// TwinCAT 3 PLC project POS_Temp_system
// ProgramVersion: 3.1.4022.3
// libraries:
//   CAA Types Extern, * (CAA Technical Workgroup)
//   Tc2_ControllerToolbox, * (Beckhoff Automation GmbH)
//   Tc2_Standard, * (Beckhoff Automation GmbH)
//   Tc2_System, * (Beckhoff Automation GmbH)
//   Tc2_Utilities, * (Beckhoff Automation GmbH)
//   Tc3_Module, * (Beckhoff Automation GmbH)
//   VisuSymbols,3.5.10.0,System
// project tree:
//   DUTs/ SeqState.TcTLEO (not stored)
//   fbBLOCKS/ fBDISCRETE_PID.TcPOU, fbSensorNoise.TcPOU, FirstOrder.TcPOU
//   / GlobalTextList.TcGTLO, PlcTask.TcTTO (not stored), Visualization Manager.TcVMO (not stored)
//   GVLs/ GVL_IO.TcGVL
//   POUs/ MAIN.TcPOU
//   PROCESSES/ HEATER_PROCESS.TcPOU, SERVO_POS.TcPOU, TANKLEVEL.TcPOU
//   VISUs/ UserInterface.TcVIS

// ---- GVLs/GVL_IO.TcGVL
{attribute 'qualified_only'}
VAR_GLOBAL
// Process parameters, variables	
	SetPoint_ServoX           :REAL;      // SetPoint X - axis
	SetPointHeater            :REAL;      // SetPoint Heater
	Output_ServoX             :REAL;      // X-axis Position
	Output_Heater             :REAL;      // Temperature Heater
	Output_Stirrer            :BOOL;      // Mixer / Stirrer 
	TankLevelSensor           :REAL;      // Tanklevel analogue sensor 
	ValveA, ValveB, ValveC    :BOOL;      // Valves
	Stirrer					  :BOOL;	  // activate stirrer
	xPushButton1              :BOOL;      // Used for test purposes 
	xPushButton2              :BOOL;      // Used for test purposes
	StartPr, StopPr           :BOOL;      // Start and Stop Process Buttons
	Level_S1,Level_S2,Level_S3:BOOL;      // Level Sensors (digital sensors)
    xGenCtrl_Error            :BOOL;      // General Error due SERVO or HEATER Control  
	//  
    noise_HeaterSensor        :BOOL;      // Sensor noise simulation on  
	noise_ServoSensor         :BOOL;      // Sensor noise simulation on          
	END_VAR

// ---- PROCESSES/TANKLEVEL.TcPOU
PROGRAM TANKLEVEL
VAR CONSTANT
	L_S1:REAL :=  5.00 ;
	L_S2:REAL := 60.00 ;
	L_S3:REAL := 80.00 ;	
END_VAR

VAR
	Plant:FirstOrder;
	//fbNoise : FB_CTRL_NOISE_GENERATOR ;
	//fbNoiseParams : ST_CTRL_NOISE_GENERATOR_PARAMS ;
	//noise_level : LREAL ;
	fill_ValveA,fill_ValveB,Drain_ValveC: BOOL;
	fbdelayOFF:TOF;
// ---	
    fbFill, fbDrain : R_TRIG;
	fbFillOff, fbDrainOff :F_TRIG;
	currConstTime: REAL := 15;
	spLevel : REAL:=0;
    SensorNoise:fbSensorNoise;
END_VAR

// Generate sensor noise
//fbNoiseParams . tCtrlCycleTime := T#10MS ;
//fbNoiseParams . tTaskCycleTime := T#10MS ;
//fbNoiseParams . fAmplitude := 1.5 ;
//fbNoise ( fManSyncValue := 1 , eMode := 2 , stParams := fbNoiseParams ) ;
//noise_level := fbNoise.fOut ;
// Valves
Fill_ValveA := GVL_IO.ValveA ;
Fill_ValveB := GVL_IO.ValveB ;
Drain_ValveC := GVL_IO.ValveC ;

fbFill(clk := ( Fill_ValveA XOR Fill_ValveB ) AND NOT Drain_ValveC ) ;
fbFillOff(clk := Fill_ValveA XOR Fill_ValveB ) ;
fbDrain(clk := Drain_ValveC );
fbDrainOff(clk := Drain_ValveC );
fbdelayOFF(IN:=(GVL_IO.ValveA OR GVL_IO.ValveB OR GVL_IO.ValveC),PT:=T#1S);

IF fbFill.Q THEN
	spLevel:=150;
	currConstTime:=15;
END_IF
IF fbFillOff.Q THEN
	spLevel:=plant.fBOut;
	
END_IF
IF fbDrain.Q THEN
	currConstTime:=5;
    spLevel:=1;	
END_IF

IF fbDrainOff.Q THEN
	spLevel := GVL_IO.TankLevelSensor ;
END_IF

Plant(fBIn:= spLevel,Gain := 1,Tconstant := currConstTime);
SensorNoise(noise_enable:=TRUE,Ampl:=1.0);
//GVL_IO.TankLevelSensor:=plant.fBOut;
GVL_IO.TankLevelSensor:=LREAL_TO_REAL(plant.fBOut +SensorNoise.noise_level);
// IF (fbdelayOFF.Q) THEN
//	GVL_IO.TankLevelSensor:=LREAL_TO_REAL(plant.fBOut +SensorNoise.noise_level);
// END_IF
GVL_IO.Level_S1:=TRUE;
GVL_IO.Level_S2:=TRUE;
GVL_IO.Level_S3:=TRUE;

IF GVL_IO.TankLevelSensor > L_S1 THEN
	GVL_IO.Level_S1:=FALSE;
END_IF
IF GVL_IO.TankLevelSensor > L_S2 THEN
	GVL_IO.Level_S2:=FALSE;
END_IF
IF GVL_IO.TankLevelSensor > L_S3 THEN
	GVL_IO.Level_S3:=FALSE;
END_IF

 //

END_PROGRAM

// ---- fbBLOCKS/FirstOrder.TcPOU
FUNCTION_BLOCK FirstOrder
VAR_INPUT
	Gain: REAL;
	Tconstant : REAL;
	fBIn   : REAL;
END_VAR
VAR_OUTPUT
	fBOut  : REAL;
END_VAR
VAR
	ssy, Sy   :REAL;
	Tsample: REAL := 0.01;
END_VAR

// This program simulates a First Order Euler Emulation
// Another way to simulate processes
// PLEASE DON'T CHANGE THE CODE IN THIS PROGRAM !
// Euler Emulation 1st Order with 0.01 sec sampletime.
sy := ( fBIn * Gain / Tconstant ) - ( fBOut / Tconstant ) ;
fBOut := fBout + ( sy * Tsample ) ;

END_FUNCTION_BLOCK

// ---- fbBLOCKS/fbSensorNoise.TcPOU
FUNCTION_BLOCK fbSensorNoise
VAR_INPUT
	noise_enable:BOOL;
	Ampl        :LREAL;
END_VAR
VAR_OUTPUT
noise_level : LREAL:=0;	
END_VAR
VAR
	fBNoise:FB_CTRL_NOISE_GENERATOR;
	fbNoiseParams: ST_CTRL_NOISE_GENERATOR_PARAMS;
END_VAR

// Generate noise for Sensors ( simulation ) 
fbNoiseParams.tCtrlCycleTime := T#10MS ;
fbNoiseParams.tTaskCycleTime := T#10MS ;
fbNoiseParams.fAmplitude := Ampl;

//
noise_level:=0;
IF Noise_enable THEN
	fbNoise ( fManSyncValue := 1 , eMode := 2 , stParams := fbNoiseParams ) ;
END_IF
noise_level:=fbNoise.fOut;

END_FUNCTION_BLOCK

// ---- fbBLOCKS/fBDISCRETE_PID.TcPOU
FUNCTION_BLOCK fBDISCRETE_PID
VAR_INPUT
	Setpoint       :REAL;   // SetPoint
    Kp             : REAL;  // Kp  Proportional gain
	Ki             : REAL;  // Ki  Integrated gain
	Kd             : REAL;  // Kd  Derivative gain
	Nfilter        : REAL;  // Lowpass Filter Coeff 
	Yprocess_value : REAL;  // Process Output
	Auto_Mode      : BOOL;  // PId enable if true (closed loop )
	MV_max_sat     : REAL;  // Maximum Saturation
	MV_min_sat     : REAL;  // Minimum Saturation
	//xExt_Error     : BOOL;  // External error 
	
END_VAR
VAR_OUTPUT
	MV_out        : REAL;    // Controller output
	Inposition    : BOOL;    //  2% Settled. is not implemented yet. 
END_VAR
VAR
	T1     : REAL :=0;
	Perr, Perr1, Perr2 : REAL ;
	deltaSetpoint :REAL;
    A,B,C  :REAL;
	MV_out1:REAL;
	Tsample:REAL := 0.01;
END_VAR

//
IF T1 = 0 THEN
	MV_out:=0;     // no bias offset  
END_IF
T1:=Tsample; 
Perr:= Setpoint - Yprocess_value; // Current error e[k]
// Check also PowerPoint Presentation module 5 
// Constant Coefficients including the Parameters Kp , Ki, Kd and Tsample
// 
//        Your PID Controller algorithm starts here
//
// A:= (Kp +Ki*(Tsample/2)+(Kd/Tsample));
// B:= (-Kp +Ki*(Tsample/2)-(2*Kd/Tsample));
// C:=  Kd/Tsample;
//
//   Mv_out:= MV_out1 + A*perr +B*perr1 + C*perr2:                                // PID Controller
//
MV_out:=  Kp * Perr;  // P-Controller 

// Update  samples 
MV_out1:= MV_out;      // MV_out[k-1] 
Perr2  := Perr1;       // e[k-2]
Perr1  := Perr;        // e[k-1]

//  PID  is not Enabled 
IF NOT Auto_Mode THEN
	MV_Out:= Setpoint;   ///  Open loop 
END_IF

//    Controller output saturation 
IF Mv_out < MV_min_sat THEN
	Mv_out:= MV_min_sat;
END_IF
IF Mv_out >  MV_max_sat THEN
	Mv_out:= MV_max_sat;
END_IF

END_FUNCTION_BLOCK

// ---- POUs/MAIN.TcPOU
PROGRAM MAIN
VAR
	PIDheater_on  : BOOL;  // PID Controller heater enabled ( Closed looop Control)
	PIDServo_on   : BOOL := TRUE;   // PID Controller heater enabled ( Closed looop Control)
	pidServo      : fBDISCRETE_PID;
	pidHeater     : fBDISCRETE_PID;
	States        : SeqState := SeqState.Ready;
	Cmd_Servo     : R_TRIG;         // For testing Servo 
	Cmd_Heater    : R_TRIG;         // For testing Heater
	Cmd_ProdStart : R_TRIG;
	Cmd_ProdStop  : R_TRIG;
	
	timerA: TP;
	TimA: F_TRIG;
END_VAR

// Handling Buttons
Cmd_ProdStart(clk:=GVL_IO.StartPr);     // Start Process
Cmd_ProdStop(clk:=GVL_IO.StopPr);       // Stop  Process
Cmd_Servo(clk:=GVL_IO.xPushButton1);    // Servo Command button for testing
Cmd_Heater(clk:=GVL_IO.xPushButton2);   // Heater Command button for testing

TimA(clk:=timerA.Q);
timerA();

// ================= START STATE SEQUENCE ======================
//
//   Your State machine program can be programmed here 
//          following an example
//
CASE States OF                       // Sequence State ( ready, etc etc etc )
	//SeqState.Ready:                  // You can change the states if you want for your own convience
	//	GVL_IO.SetPointHeater:= 75;  // Setpoint heater 75 degrees Celsius. 
//	
//SeqState.Fill_A:
		//GVL_IO .ValveA:=TRUE;    //  Open Valve A 	
//	
//

	SeqState.Ready:
	IF GVL_IO.StartPr = TRUE AND GVL_IO.StopPr = FALSE THEN
		GVL_IO.SetPointHeater := 75;
		States := SeqState.Fill_A;
	END_IF
	
	SeqState.TO_INIT:
	GVL_IO.SetPointHeater := 0;
	IF GVL_IO.Output_ServoX > -0.4 AND GVL_IO.Output_ServoX < 0.6 THEN
		PIDServo_on := FALSE;
	ELSE
		GVL_IO.SetPoint_ServoX := 0;
		PIDServo_on := TRUE;
	END_IF
	
	IF (GVL_IO.Output_Heater > 0 AND GVL_IO.Output_Heater < 1.5) AND GVL_IO.Level_S1 = TRUE AND (GVL_IO.Output_ServoX > -0.4 AND GVL_IO.Output_ServoX < 0.6) THEN
		States := SeqState.Ready;
	END_IF
	
	SeqState.Fill_A:
	GVL_IO.ValveA := TRUE;
	
	IF GVL_IO.Level_S2 = FALSE THEN
		GVL_IO.ValveA := FALSE;
		States := SeqState.Fill_B;
	END_IF
	
	SeqState.Fill_B:
	GVL_IO.ValveB := TRUE;
	PIDheater_on := TRUE;
	GVL_IO.Stirrer := TRUE;
	IF GVL_IO.Level_S3 = FALSE THEN
		GVL_IO.ValveB := FALSE;
		States := SeqState.Heating;
	END_IF
	
	SeqState.Heating:
	IF GVL_IO.Output_Heater > 73.5 AND GVL_IO.Output_Heater < 76.5 THEN
		// turn on timer
		timerA(IN:= TRUE, PT:= T#20S);
		
		// check timer
		IF TimA.Q THEN	
			States := SeqState.ToUnload;
		END_IF
		
	END_IF
	
	SeqState.ToUnload:
	GVL_IO.SetPoint_ServoX := 30;
	PIDServo_on := TRUE;
	
	IF GVL_IO.Output_ServoX > 29.4 AND GVL_IO.Output_ServoX < 30.6 THEN
		PIDServo_on := FALSE;
		PIDheater_on := FALSE;
		States := SeqState.Drain_1;
	END_IF
	
	
	SeqState.Drain_1:
	GVL_IO.ValveC := TRUE;
	IF GVL_IO.Level_S2 = TRUE THEN
		States := SeqState.Drain_2;
	END_IF
	
	SeqState.Drain_2:
	GVL_IO.Stirrer := FALSE;
	IF GVL_IO.Level_S1 = TRUE THEN
		GVL_IO.ValveC := FALSE;
		States := SeqState.TO_INIT;
	END_IF

	
END_CASE
//
//
// ================ END of the STATE SEQUENCES      =====================
// 
// =====   Executing the PID Controllers for  Position and Heater.   =======
//
// *************  Servo with P- Controller only  **************
//
IF (Cmd_Servo.Q ) THEN
	pidServo.Setpoint:=GVL_IO.SetPoint_ServoX;  // Setpoint Servo
END_IF

pidServo.Kp:= 1;       //  Kp parameter
// pidServo.Ki:= xxx ; //  Ki parameter
// pidServo.Kd:= xxx ; //  Kd parameter 

pidServo.MV_max_sat:=  10;   // Maximum output PID to protect the Servo
pidServo.MV_min_sat:= -10;   // Minimum output PID    ,,     ,,
pidServo.Yprocess_value:= LREAL_TO_REAL(SERVO_POS.Tf_SERVO_Output);
//
pidServo(Auto_Mode:=PIDServo_on,MV_out=>SERVO_POS.Tf_SERVO_Input);  // Calling PID function Heater

// *************   Heater with P- Controller only   **********************
//
IF Cmd_Heater.Q THEN
   pidHeater.Setpoint:=GVL_IO.SetPointHeater;	
END_IF
pidHeater.Kp:= 0.5;           //  Kp parameter
// pidHeater.Ki:= xx ;       //  Ki parameter     
// pidHeater.Kd:= xx ;       //  Kd parameter      
pidHeater.MV_max_sat:= 150;  // Maximum output PID to protect the Heater
pidHeater.MV_min_sat:= -10;  // Minimum output PID ,,     ,,
pidHeater.Yprocess_value:=LREAL_TO_REAL( HEATER_PROCESS.Tf_Heater_Output);
pidHeater(Auto_Mode:= PIDheater_on,MV_out=>HEATER_PROCESS.Tf_Heater_Input);  // Calling PID function Heater

END_PROGRAM

// ---- PROCESSES/SERVO_POS.TcPOU
PROGRAM SERVO_POS
VAR CONSTANT
	nTfOrder : USINT := 2;
	nNumOrder : USINT :=2;
	nDenOrder : USINT :=2;
END_VAR
VAR_INPUT
	Tf_SERVO_Input:LREAL;
END_VAR
VAR_OUTPUT
	Tf_SERVO_Output:LREAL;
END_VAR
VAR
	aNumArray    : ARRAY[0..nNumOrder] OF FLOAT; //numerator
	aDenArray    : ARRAY[0..nDenOrder] OF FLOAT; //denumerator
	aStructTfData: ARRAY[0..nTfOrder]  OF ST_CTRL_TRANSFERFUNCTION_1_DATA;
	eMode        : E_CTRL_MODE;
	stParams     : ST_CTRL_TRANSFERFUNCTION_1_PARAMS;
	eErrorId     : E_CTRL_ERRORCODES;
	bError       : BOOL;
	fbServoX_Tf  : FB_CTRL_TRANSFERFUNCTION_1;
	bInit        : BOOL := TRUE;
	bPosError    :BOOL;
	fb_Output    : LREAL;
	Servo_ERR    : R_TRIG;
    SensorNoise  :fbSensorNoise;
END_VAR

// IA _Cs4  2019
// O.E Figaroa
// This program simulates a First Order DC Servo with an Integrator
// PLEASE DON'T CHANGE THE CODE IN THIS PROGRAM !
// Transferfunction Servo Motor X s-domain
//              20
//  Gc =    -----------   [ Theta/u]    and u is proportional to angular position [Theta]
//           0.5s^2 + s 
//
//= = Discrete or z-domain with  Ts = 0.01 s = = 
//          short format
//        0.001987 z + 0.001974
// Gd =  ----------------------   with Ts=0.01 s
//        z^2 - 1.98 z + 0.9802       
// 
//// coefficients obtained by Matlab in long format:
//
// numz =  [0   0.001986733067553   0.001973532271096]     
// denz =  [1.000000000000000 -1.980198673306755   0.980198673306755]
// ==

//========================================
IF bInit THEN
// = numerator ===
aNumArray[0] := 0.001973532271096; 
aNumArray[1] := 0.001986733067553; 
aNumArray[2] := 0.000;
// = denumerator
aDenArray[0] := 0.980198673306755;
aDenArray[1] := -1.980198673306755;
aDenArray[2] := 1.0;
stParams.tTaskCycleTime := T#10MS;
stParams.tCtrlCycleTime := T#10MS;
stParams.nOrderOfTheTransferfunction := nTfOrder;
eMode := eCTRL_MODE_ACTIVE;
bInit := FALSE;
END_IF
stParams.pNumeratorArray_ADR := ADR(aNumArray);
stParams.nNumeratorArray_SIZEOF := SIZEOF(aNumArray);
stParams.pDenominatorArray_ADR := ADR(aDenArray);
stParams.nDenominatorArray_SIZEOF := SIZEOF(aDenArray);
stParams.pTransferfunction1Data_ADR := ADR(aStructTfData);
stParams.nTransferfunction1Data_SIZEOF := SIZEOF(aStructTfData);

// Execute TF 

fbServoX_Tf (fIn :=Tf_SERVO_Input,
eMode := eMode,
stParams := stParams,
fOut => fb_Output,
eErrorId => eErrorId,
bError => bError);
// Sensor Noises
SensorNoise(Ampl:=0.3);
SensorNoise(noise_enable:=GVL_IO.noise_ServoSensor);
Tf_SERVO_Output:=fb_Output+ SensorNoise.noise_level ;
GVL_IO.Output_ServoX:=LREAL_TO_REAL(Tf_SERVO_Output);	

Servo_ERR(CLK:=(ABS(GVL_IO.Output_ServoX) > 50),Q=>GVL_IO.xGenCtrl_Error);

END_PROGRAM

// ---- PROCESSES/HEATER_PROCESS.TcPOU
PROGRAM HEATER_PROCESS
VAR CONSTANT
	nTfOrder : USINT := 2;
	nNumOrder : USINT :=2;
	nDenOrder : USINT :=2;
END_VAR
VAR_INPUT
	Tf_Heater_Input : LREAL;
END_VAR
VAR_OUTPUT
	Tf_Heater_Output : LREAL;
END_VAR
VAR
	aNumArray        : ARRAY[0..nNumOrder] OF FLOAT; //numerator
	aDenArray        : ARRAY[0..nDenOrder] OF FLOAT; //denumerator
	aStructTfData    : ARRAY[0..nTfOrder]  OF ST_CTRL_TRANSFERFUNCTION_1_DATA;
	eMode            : E_CTRL_MODE;
	stParams         : ST_CTRL_TRANSFERFUNCTION_1_PARAMS;
	eErrorId         : E_CTRL_ERRORCODES;
	bError           : BOOL;
	fbHeater_Tf      : FB_CTRL_TRANSFERFUNCTION_1;
	bInit            : BOOL := TRUE;
	fb_Output        : LREAL;
	SensorNoise      :fbSensorNoise;	 
END_VAR

// IA _Cs4  2019
// O.E Figaroa
// This program simulates a Second Order Process aka Heater Process.
// PLEASE DON'T CHANGE THE CODE IN THIS PROGRAM !
// Transferfunction Heater
//                  5
///  G(s)=  ---------------------    [ Temp / Temp ]
//          256 s^2 + 100 s + 5
//= = = = = = = = = = = = = = = = 
// Discrete transfer function of the Heater
//
//
//          9.753E-07 z + 9.74E-07
// G(z)=  ----------------------
//          z^2 - 1.996 z + 0.9961
//
// Obtained coefficients in long formats for accuracy purposes
//
// numerator =    1.0e-06 * [0   0.975292016341129   0.974022931328863]
// denumerator = [1.000000000000000  -1.996099420155170   0.996101369470118]

IF bInit THEN
// = numerator ===
aNumArray[0] := 0.974022931328863 * 1E-06;
aNumArray[1] := 0.975292016341129 * 1E-06;
aNumArray[2] := 0.000;
// = denumerator
aDenArray[0] := 0.996101369470118;
aDenArray[1] := -1.996099420155170;
aDenArray[2] := 1.00000;
// 

stParams.tTaskCycleTime := T#10MS;
stParams.tCtrlCycleTime := T#10MS;
stParams.nOrderOfTheTransferfunction := nTfOrder;
eMode := eCTRL_MODE_ACTIVE;
bInit := FALSE;
END_IF

stParams.pNumeratorArray_ADR := ADR(aNumArray);
stParams.nNumeratorArray_SIZEOF := SIZEOF(aNumArray);
stParams.pDenominatorArray_ADR := ADR(aDenArray);
stParams.nDenominatorArray_SIZEOF := SIZEOF(aDenArray);
stParams.pTransferfunction1Data_ADR := ADR(aStructTfData);
stParams.nTransferfunction1Data_SIZEOF := SIZEOF(aStructTfData);
// Execute TF 
fbHeater_Tf (fIn := Tf_Heater_Input,
eMode := eMode,
stParams := stParams,
fOut => fb_Output,
eErrorId => eErrorId,
bError => bError);
//
//
SensorNoise(Ampl:=1.5);
SensorNoise(noise_enable:=GVL_IO.noise_HeaterSensor) ; // Sensor Noise 
Tf_Heater_Output:= fb_Output + SensorNoise.noise_level;

GVL_IO.Output_Heater:=LREAL_TO_REAL(Tf_Heater_Output);
IF fbHeater_Tf.fOut < 0 THEN
	GVL_IO.Output_Heater:=0;
END_IF

END_PROGRAM

// ---- GlobalTextList.TcGTLO
TEXTLIST GlobalTextList
  249 = '%.1d'
  0 = '%.1f'
  112 = '%.2f'
  438 = '%d'
  228 = 'Auto-Mode Closed loopServo'
  47 = 'Auto-Mode Heater'
  280 = 'Auto-Mode Servo'
  694 = 'Auto-Modee Servo'
  528 = 'Closed loop Servo'
  753 = 'Drain Position'
  70 = 'Heater  Sensor noise enabled'
  338 = 'Heater noise Sensor enabled'
  601 = 'Home'
  167 = 'Outlet'
  445 = 'Output Heater   %.2f'
  952 = 'Output Heater  %.2f'
  735 = 'Output PID  %.2f'
  160 = 'Output Servo   %.2f'
  65 = 'Output Servo  %.2f'
  940 = 'Overshoot'
  350 = 'Overshoot= 30'
  17 = 'PID-Enable'
  786 = 'PID-Enable Heater'
  168 = 'PID-Enable Servo'
  520 = 'Position %s'
  468 = 'Position = 0'
  917 = 'Position = 30'
  409 = 'Position and Temperature Control in Batch Process'
  224 = 'Position and Temperature Control in Batch Processes'
  93 = 'Response %s'
  81 = 'Response X -axis %s'
  617 = 'Response X -axis:   %s'
  12 = 'Response Y -axis %s'
  134 = 'Response Y -axis:   %s'
  150 = 'Servo Error'
  621 = 'Servo Running CCW'
  837 = 'Servo Sensor  noise enabled'
  147 = 'Setpoint %.2f'
  636 = 'SetPoint %s'
  401 = 'Setpoint Heater   %.2f'
  318 = 'Setpoint Heater  %.2f'
  352 = 'Setpoint Servo   %.2f'
  905 = 'Setpoint Servo  %.2f'
  368 = 'SetPoint: %d'
  75 = 'SetPoint: %s'
  637 = 'SP Heater cmd'
  808 = 'SP Servo cmd'
  97 = 'START'
  126 = 'STOP'
  527 = 'Tank'
  652 = 'TANK'
  534 = 'Tank %.2f'
  946 = 'Tanklevel %.2f'
  181 = 'Tanklevel Sensor:    %.2f'
  276 = 'Tanklevel:    %.2f'
  119 = 'Unload  Position'
  471 = 'WALL'
  434 = 'Wall HIT !'
END_TEXTLIST

// ---- VISUs/UserInterface.TcVIS
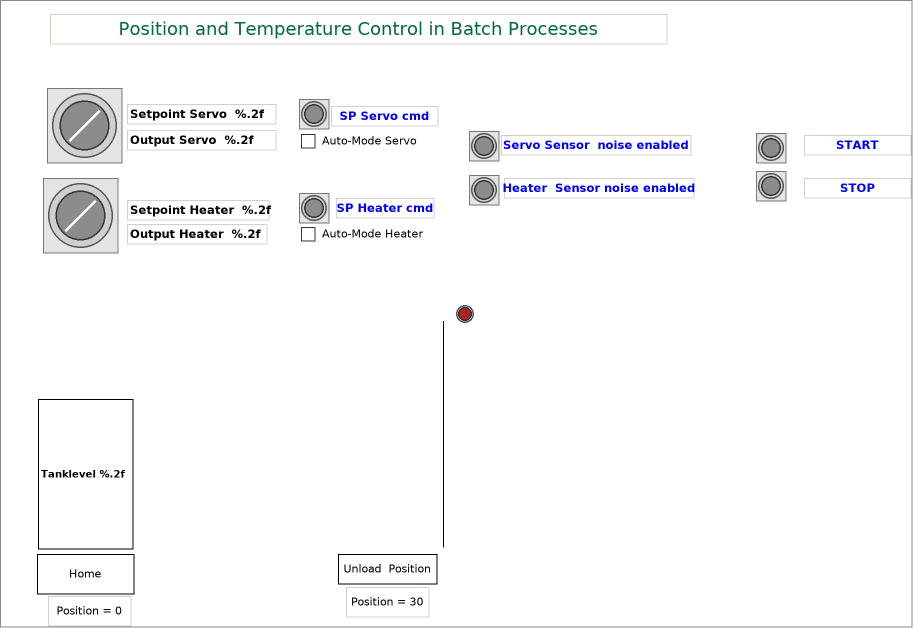
VISUALIZATION UserInterface  // 913x628
    PushSwitch (299,99 30x30), variable: GVL_IO.xPushButton1, behaviour: TAP, style: Switch-PushSwitch-Gray
    Potentiometer360 (47,88 75x75), variable: GVL_IO.SetPoint_ServoX, style: Potentiometer-Potentiometer360-Gray, scale format: %d, scale 0..60
        p2431819421: Outside
    Textfield (127,104 149x20), "Setpoint Servo %.2f", text variable: GVL_IO.SetPoint_ServoX
    Textfield (127,130 149x20), "Output Servo %.2f", text variable: GVL_IO.Output_ServoX
    Potentiometer360 (43,178 75x75), variable: GVL_IO.SetPointHeater, style: Potentiometer-Potentiometer360-Gray, scale format: %d, scale 15..115
        p2431819421: Outside
    PushSwitch (299,193 30x30), variable: GVL_IO.xPushButton2, behaviour: TAP, style: Switch-PushSwitch-Gray
    Textfield (127,200 142x20), "Setpoint Heater %.2f", text variable: GVL_IO.SetPointHeater
    Textfield (127,224 140x20), "Output Heater %.2f", text variable: GVL_IO.Output_Heater
    Rectangle (37,554 97x40), "Home"
    Rectangle (338,554 99x30), "Unload Position"
    Textfield (346,587 83x30), "Position = 30"
    Textfield (48,596 83x30), "Position = 0"
    Rectangle (38,399 95x150), "Tanklevel %.2f", text variable: GVL_IO.TankLevelSensor
        p3560616238: GVL_IO.Output_ServoX * 10
    Textfield (336,198 98x20), "SP Heater cmd"
    Textfield (331,106 107x20), "SP Servo cmd"
    Textfield (50,14 617x30), "Position and Temperature Control in Batch Processes"
    Checkbox (299,224 125x20), "Auto-Mode Heater", variable: MAIN.PIDheater_on
    Checkbox (299,131 195x20), "Auto-Mode Servo", variable: MAIN.PIDServo_on
    Line (443,321) (443,547)
    Lamp1 (455,304 20x20), variable: (GVL_IO.Output_ServoX>31), style: Lamp-Lamp1-Red
    PushSwitch (469,175 30x30), variable: GVL_IO.noise_HeaterSensor, behaviour: TOGGLE, style: Switch-PushSwitch-Gray
    Textfield (504,178 190x20), "Heater Sensor noise enabled"
    PushSwitch (469,131 30x30), variable: GVL_IO.noise_ServoSensor, behaviour: TOGGLE, style: Switch-PushSwitch-Gray
    Textfield (501,135 190x20), "Servo Sensor noise enabled"
    PushSwitch (756,133 30x30), variable: GVL_IO.StartPr, behaviour: TOGGLE, style: Switch-PushSwitch-Gray
    PushSwitch (756,171 30x30), variable: GVL_IO.StopPr, behaviour: TOGGLE, style: Switch-PushSwitch-Gray
    Textfield (804,135 107x20), "START"
    Textfield (804,178 107x20), "STOP"
END_VISUALIZATION
